// TIA Portal V20 export
TYPE "typeFDoorUnlockOutput"
// stored: Access Published, IsFailsafeCompliant true, Namespace Safety
   STRUCT
      autoSpliceDoorUnlock : Bool;   // F Door Unlock Cmd Status
      unwinderMainDoorUnlock : Bool;   // F Door Unlock Cmd Status
      unwinderTopDoorUnlock : Bool;   // F Door Unlock Cmd Status
      unwinderBtmDoorUnlock : Bool;   // F Door Unlock Cmd Status
      stackTableDoorUnlock : Bool;   // F Door Unlock Cmd Status
      jrWinderDoorUnlock : Bool;   // F Door Unlock Cmd Status
      anodeWasteDoorUnlock : Bool;   // F Door Unlock Cmd Status
      stackTableRearDoorUnlock : Bool;   // F Door Unlock Cmd Status
      cathodeWasteDoorUnlock : Bool;   // F Door Unlock Cmd Status
      unwinderRearDoorUnlock : Bool;   // F Door Unlock Cmd Status
   END_STRUCT;
END_TYPE
